FUNCTION MinDistanceValue : lreal
VAR_INPUT
	rowValue:LREAL;
	refValue:LREAL;
END_VAR
VAR
	rowValueAdd2Pi:LREAL;
	rowValueReduce2Pi:LREAL;
	distance:LREAL;
END_VAR

rowValueAdd2Pi:=rowValue+2*pi;
rowValueReduce2Pi:=rowValue-2*pi;
distance:=Min3Value(ABS(rowValue-refValue),ABS(rowValueAdd2Pi-refValue),ABS(rowValueReduce2Pi-refValue));
IF distance=ABS(rowValue-refValue) THEN
	MinDistanceValue:=rowValue;
ELSIF distance=ABS(rowValueAdd2Pi-refValue) THEN
	MinDistanceValue:=rowValueAdd2Pi;
ELSE
	MinDistanceValue:=rowValueReduce2Pi;
END_IF

END_FUNCTION

(* stored: Version 1.1.0.1, ProductVersion 3.1.4024.2
   POU MinDistanceValue: Id {96b9a079-1681-4836-854d-2ee02e553fad}, SpecialFunc None *)
